(* IEC 61131-3 sources: LAxisCtrl/src/blocks (part 3) *)

                            ELSIF (_instCamIn.Error = TRUE) THEN
                                // Errorhandling
                                _status := AxisStatus#ERR_MC_CAMIN;
                                _statusText := STRING#'ERR_MC_CAMIN';
                                _errorAutoCleared := TRUE;
                                _diagnostics.subfunctionStatus := _instCamIn.ErrorId;
                                _subfunctionStatus := _instCamIn.ErrorId;
                                _diagnostics.basicMotionState := _basicMotionState;
                                _state := AXIS_STOP_ON_ERROR_SELECTION;
                                _basicMotionState := NO_SELECTION;
                            // ELSE
                            //   ; // Command selected
                            END_IF;

                            // Write MC_Command outputs to internal variable
                            _exeOfBasicMotion := 16#0;
                            _exeOfBasicMotion.%X0 := _instCamIn.Busy;
                            IF (_applicationMode = APPLICATION_MODE_ONCE) THEN
                                _exeOfBasicMotion.%X1 := _instCamIn.EndOfProfile;
                            END_IF;
                            _exeOfBasicMotion.%X2 := _instCamIn.CommandAborted;
                            _exeOfBasicMotion.%X3 := _instCamIn.Error;
                            _exeOfBasicMotion.%X6 := _instCamIn.StartSync;
                            _exeOfBasicMotion.%X7 := _instCamIn.InSync;
                            _exeOfBasicMotion.%X8 := _instCamIn.EndOfProfile;

                        GEAR_OUT_CAM_OUT_SELECTED:

                        // Firstcycle of command
                        IF (_firstCycleBasicMotion = TRUE) THEN
                            _applicativeBasicMotionError := FALSE;
                            _firstCycleBasicMotion := FALSE;

                            // Reset CAM_OUT command
                            _instCamOut(Slave := _refSyncAxis^,
                                        Execute := FALSE,
                                        SlavePosition := config.gearOutCamOut.slavePosition,
                                        SyncProfileReference := config.gearOutCamOut.syncProfileReference,
                                        MasterStopDistance := config.gearOutCamOut.masterStopDistance,
                                        Deceleration := config.gearOutCamOut.deceleration,
                                        Jerk := config.gearOutCamOut.jerk,
                                        SyncOutDirection := config.gearOutCamOut.syncOutDirection);

                            // Reset GEAR_OUT command
                            _instGearOut(Slave := _refSyncAxis^,
                                         Execute := FALSE,
                                         SlavePosition := config.gearOutCamOut.slavePosition,
                                         SyncProfileReference := config.gearOutCamOut.syncProfileReference,
                                         MasterStopDistance := config.gearOutCamOut.masterStopDistance,
                                         Deceleration := config.gearOutCamOut.deceleration,
                                         Jerk := config.gearOutCamOut.jerk,
                                         SyncOutDirection := config.gearOutCamOut.syncOutDirection);

                            CASE config.gearOutCamOut.gearOutCamOutMode OF
                                SYNCOUT_MODE_AUTOMATIC,
                                SYNCOUT_MODE_GEAROUT,
                                SYNCOUT_MODE_CAMOUT:
                                    // Get axis waiting function state
                                    IF (_typeAxis = SYNC_AXIS) THEN
                                        IF (_waitingFunctionStateAbortAutomatic < 0) // < 0: Automatic abort of waiting sync commands disabled
                                        THEN
                                            // Read waiting function state of axis
                                            _waitingFunctionState := _refSyncAxis^.StatusSynchronizedMotion.WaitingFunctionState;
                                        ELSE
                                            // Waiting function state already read out
                                            _waitingFunctionState := _waitingFunctionStateAbortAutomatic;
                                        END_IF;
                                        // Read function state of axis
                                        _functionState := _refSyncAxis^.StatusSynchronizedMotion.FunctionState;
                                    END_IF;

                                    _gearAndCamOutMode := config.gearOutCamOut.gearOutCamOutMode;
                                    _syncOutState := SYNCOUT_STATE_CHECK_WAITING; // Set next state

                                ELSE
                                    // Errorhandling - Invalid mode
                                    _status := AxisStatus#ERR_INVALID_GEAROUT_CAMOUT_MODE;
                                    _statusText := STRING#'ERR_INVALID_GEAROUT_CAMOUT_MODE';
                                    _errorAutoCleared := TRUE;
                                    _diagnostics.subfunctionStatus := WORD#0000;
                                    _subfunctionStatus := AxisStatus#STATUS_NO_CALL;
                                    _applicativeBasicMotionError := TRUE;
                                    // Set next state
                                    _state := AXIS_STOP_ON_ERROR_SELECTION;
                                    _basicMotionState := NO_SELECTION;
                            END_CASE;
                        END_IF;

                        IF (_applicativeBasicMotionError = FALSE) THEN
                            CASE _syncOutState OF
                                // ===========================================================
                                SYNCOUT_STATE_CHECK_WAITING:

                                    CASE _gearAndCamOutMode OF
                                        SYNCOUT_MODE_GEAROUT:
                                            CASE _waitingFunctionStateAbortAutomatic OF
                                                WFS_FS_CAMIN:
                                                    // Abort waiting camming in advance
                                                    _instCamOut.SyncProfileReference := CANCEL_ONLY_WAITING_GEARING_CAMMING;
                                                    _syncOutState := SYNCOUT_STATE_CAMOUT_WAITING_BUSY; // Set next state

                                                WFS_FS_GEARINPOS:
                                                    CASE config.gearOutCamOut.syncProfileReference OF
                                                        CANCEL_ONLY_WAITING_GEARING_CAMMING:
                                                            // Only gearOut - Set next state
                                                            _syncOutState := SYNCOUT_STATE_CHECK_ACTIVE;
                                                    ELSE
                                                        CASE _functionState OF
                                                            WFS_FS_GEARIN,
                                                            WFS_FS_GEARINPOS:
                                                                // Active gearing function
                                                                _syncOutState := SYNCOUT_STATE_CHECK_ACTIVE; // Set next state
                                                        ELSE
                                                            // Abort waiting gearing in advance
                                                            _instGearOut.SyncProfileReference := CANCEL_ONLY_WAITING_GEARING_CAMMING;
                                                            _syncOutState := SYNCOUT_STATE_GEAROUT_WAITING_BUSY; // Set next state
                                                        END_CASE;
                                                    END_CASE;

                                            ELSE
                                                // Only gearOut - Set next state
                                                _syncOutState := SYNCOUT_STATE_CHECK_ACTIVE;
                                            END_CASE;

                                        SYNCOUT_MODE_CAMOUT:
                                            CASE _waitingFunctionStateAbortAutomatic OF
                                                WFS_FS_GEARINPOS: // Waiting
                                                    // Abort waiting gearing in advance
                                                    _instGearOut.SyncProfileReference := CANCEL_ONLY_WAITING_GEARING_CAMMING;
                                                    _syncOutState := SYNCOUT_STATE_GEAROUT_WAITING_BUSY; // Set next state

                                                WFS_FS_CAMIN: // Waiting
                                                    CASE config.gearOutCamOut.syncProfileReference OF
                                                        CANCEL_ONLY_WAITING_GEARING_CAMMING:
                                                            // Only gearOut - Set next state
                                                            _syncOutState := SYNCOUT_STATE_CHECK_ACTIVE;
                                                    ELSE
                                                        CASE _functionState OF
                                                            WFS_FS_CAMIN: // Active
                                                                _syncOutState := SYNCOUT_STATE_CHECK_ACTIVE; // Set next state
                                                        ELSE
                                                            // Abort waiting camming in advance
                                                            _instCamOut.SyncProfileReference := CANCEL_ONLY_WAITING_GEARING_CAMMING;
                                                            _syncOutState := SYNCOUT_STATE_CAMOUT_WAITING_BUSY; // Set next state
                                                        END_CASE;
                                                    END_CASE;
                                            ELSE
                                                // Only camOut - Set next state
                                                _syncOutState := SYNCOUT_STATE_CHECK_ACTIVE;
                                            END_CASE;

                                        SYNCOUT_MODE_AUTOMATIC:
                                            CASE _waitingFunctionState OF
                                                WFS_FS_GEARINPOS, // Waiting
                                                WFS_FS_GEAROUT: // Waiting
                                                    CASE _functionState OF
                                                        WFS_FS_GEARIN, // Active
                                                        WFS_FS_GEARINPOS: // Active
                                                            ; // Gearing active - Waiting gearInPos will be aborted with MC_GEAROUT

                                                        WFS_FS_GEAROUT:
                                                            IF (_waitingFunctionStateAbortAutomatic < 0) THEN
                                                                ; // Automatic abort of waiting sync commands disabled
                                                            ELSE
                                                                // Automatic abort of waiting sync commands enabled - Separate call of MC_GearOut instruction is required
                                                                _instGearOut.SyncProfileReference := CANCEL_ONLY_WAITING_GEARING_CAMMING;
                                                            END_IF;
                                                    ELSE
                                                        _instGearOut.SyncProfileReference := CANCEL_ONLY_WAITING_GEARING_CAMMING;
                                                    END_CASE;
                                                    _functionState := -1;// Function state has to be updated at next use
                                                    _syncOutState := SYNCOUT_STATE_GEAROUT_WAITING_BUSY; // Set next state

                                                WFS_FS_CAMIN,  // Waiting
                                                WFS_FS_CAMOUT:  // Waiting
                                                    CASE _functionState OF
                                                        WFS_FS_CAMIN: // Active
                                                            ; // CamIn Active - Waiting CamIn will be aborted with MC_CAMOUT

                                                        WFS_FS_CAMOUT: // Active
                                                            IF (_waitingFunctionStateAbortAutomatic < 0) THEN
                                                                ; // Automatic abort of waiting sync commands disabled
                                                            ELSE
                                                                // Automatic abort of waiting sync commands enabled - Separate call of MC_CamOut instruction is required
                                                                _instCamOut.SyncProfileReference := CANCEL_ONLY_WAITING_GEARING_CAMMING;
                                                            END_IF;
                                                    ELSE
                                                        _instCamOut.SyncProfileReference := CANCEL_ONLY_WAITING_GEARING_CAMMING;
                                                    END_CASE;
                                                    _functionState := -1;// Function state has to be updated at next use
                                                    _syncOutState := SYNCOUT_STATE_CAMOUT_WAITING_BUSY; // Set next state

                                        ELSE
                                            // No waiting synchronous operation
                                            _syncOutState := SYNCOUT_STATE_CHECK_ACTIVE; // Set next state
                                        END_CASE;
                                    END_CASE;
                                    tempStateChangeActive := TRUE;

                                // ===========================================================
                                SYNCOUT_STATE_CHECK_ACTIVE:

                                    _instGearOut.SyncProfileReference := config.gearOutCamOut.syncProfileReference;
                                    _instCamOut.SyncProfileReference := config.gearOutCamOut.syncProfileReference;

                                    CASE _gearAndCamOutMode OF
                                        SYNCOUT_MODE_GEAROUT:
                                            _syncOutState := SYNCOUT_STATE_GEAROUT_ACTIVE_BUSY; // Set next state

                                        SYNCOUT_MODE_CAMOUT:
                                            _syncOutState := SYNCOUT_STATE_CAMOUT_ACTIVE_BUSY; // Set next state

                                        SYNCOUT_MODE_AUTOMATIC:
                                            CASE config.gearOutCamOut.syncProfileReference OF
                                                CANCEL_ONLY_WAITING_GEARING_CAMMING:
                                                    // No active synchronous operation
                                                    _syncOutState := SYNCOUT_STATE_DONE; // Set next state
                                            ELSE
                                                // Update function state of axis
                                                IF (_typeAxis = SYNC_AXIS) THEN
                                                    IF (_functionState < 0) THEN
                                                        _functionState := _refSyncAxis^.StatusSynchronizedMotion.FunctionState;
                                                    END_IF;
                                                END_IF;

                                                CASE _functionState OF
                                                    WFS_FS_GEAROUT,   // Active - Leads to error of MC_Instruction
                                                    WFS_FS_GEARIN,    // Active
                                                    WFS_FS_GEARINPOS: // Active
                                                        // Active gearing function
                                                        _syncOutState := SYNCOUT_STATE_GEAROUT_ACTIVE_BUSY; // Set next state

                                                    WFS_FS_CAMOUT, // Active - Leads to error of MC_Instruction
                                                    WFS_FS_CAMIN:  // Active
                                                        // Active camming function
                                                        _syncOutState := SYNCOUT_STATE_CAMOUT_ACTIVE_BUSY; // Set next state

                                                ELSE
                                                    // No active synchronous operation
                                                    _syncOutState := SYNCOUT_STATE_DONE; // Set next state
                                                END_CASE;
                                            END_CASE;

                                    END_CASE;
                                    tempStateChangeActive := TRUE;

                                // ===========================================================
                                SYNCOUT_STATE_GEAROUT_WAITING_BUSY,
                                SYNCOUT_STATE_GEAROUT_ACTIVE_BUSY:

                                    // Call MC_Instruction
                                    _instGearOut(Slave := _refSyncAxis^,
                                                Execute := TRUE);

                                    IF _instGearOut.Done THEN
                                        CASE _syncOutState OF
                                            SYNCOUT_STATE_GEAROUT_WAITING_BUSY:
                                            // Set next state
                                            _syncOutState := SYNCOUT_STATE_CHECK_ACTIVE;
                                            tempStateChangeActive := TRUE;

                                            SYNCOUT_STATE_GEAROUT_ACTIVE_BUSY:
                                            _syncOutState := SYNCOUT_STATE_DONE; // Set next state

                                        END_CASE;
                                        // Reset MC_Instruction
                                        _instGearOut(Slave := _refSyncAxis^,
                                                    Execute := FALSE);

                                    ELSIF _instGearOut.CommandAborted THEN
                                        _syncOutState := SYNCOUT_STATE_ABORTED; // Set next state
                                    END_IF;

                                // ===========================================================
                                SYNCOUT_STATE_CAMOUT_WAITING_BUSY,
                                SYNCOUT_STATE_CAMOUT_ACTIVE_BUSY:

                                    // Call MC_Instruction
                                    _instCamOut(Slave := _refSyncAxis^,
                                                Execute := TRUE);

                                    IF _instCamOut.Done THEN
                                        CASE _syncOutState OF
                                            SYNCOUT_STATE_CAMOUT_WAITING_BUSY:
                                                // Set next state
                                                _syncOutState := SYNCOUT_STATE_CHECK_ACTIVE;
                                                tempStateChangeActive := TRUE;

                                            SYNCOUT_STATE_CAMOUT_ACTIVE_BUSY:
                                                _syncOutState := SYNCOUT_STATE_DONE; // Set next state

                                        END_CASE;

                                        // Reset MC_Instruction
                                        _instCamOut(Slave := _refSyncAxis^,
                                                    Execute := FALSE);

                                    ELSIF _instCamOut.CommandAborted THEN
                                        _syncOutState := SYNCOUT_STATE_ABORTED; // Set next state
                                    END_IF;

                                // ===========================================================
                                SYNCOUT_STATE_DONE,
                                SYNCOUT_STATE_ABORTED,
                                SYNCOUT_STATE_ERROR:

                                    IF NOT _basicCommand.%X11 THEN
                                        // Return to NO_SELECTION if command finished
                                        _basicMotionState := NO_SELECTION;
                                    END_IF;

                            END_CASE;

                            IF _instGearOut.Error THEN
                                // Errorhandling
                                _status := AxisStatus#ERR_MC_GEAROUT;
                                _statusText := STRING#'ERR_MC_GEAROUT';
                                _errorAutoCleared := TRUE;
                                _diagnostics.subfunctionStatus := _instGearOut.ErrorId;
                                _subfunctionStatus := _instGearOut.ErrorId;
                                _diagnostics.basicMotionState := _basicMotionState;
                                _state := AXIS_STOP_ON_ERROR_SELECTION;
                                _basicMotionState := NO_SELECTION;

                                _syncOutState := SYNCOUT_STATE_ERROR; // Set next state

                            ELSIF _instCamOut.Error THEN
                                // Errorhandling
                                _status := AxisStatus#ERR_MC_CAMOUT;
                                _statusText := STRING#'ERR_MC_CAMOUT';
                                _errorAutoCleared := TRUE;
                                _diagnostics.subfunctionStatus := _instCamOut.ErrorId;
                                _subfunctionStatus := _instCamOut.ErrorId;
                                _diagnostics.basicMotionState := _basicMotionState;
                                _state := AXIS_STOP_ON_ERROR_SELECTION;
                                _basicMotionState := NO_SELECTION;

                                _syncOutState := SYNCOUT_STATE_ERROR; // Set next state
                            END_IF;

                            // Write MC_Command outputs to internal variable
                            _exeOfBasicMotion := 16#0;
                            _exeOfBasicMotion.%X0 := _syncOutState < SYNCOUT_STATE_DONE; // 7
                            _exeOfBasicMotion.%X1 := _syncOutState = SYNCOUT_STATE_DONE; // 7
                            _exeOfBasicMotion.%X2 := _syncOutState = SYNCOUT_STATE_ABORTED; // 8
                            _exeOfBasicMotion.%X3 := _syncOutState = SYNCOUT_STATE_ERROR; // 9
                            _exeOfBasicMotion.%X6 := _instCamOut.StartSyncOut OR _instGearOut.StartSyncOut;
                        END_IF;

                    ELSE
                        // Errorhandling
                        _status := AxisStatus#ERR_UNDEFINED_BASIC_MOTION_STATE;
                        _statusText := STRING#'ERR_UNDEFINED_BASIC_MOTION_STATE';
                        _errorUserCleared := TRUE;
                        _diagnostics.subfunctionStatus := WORD#0000;
                        _subfunctionStatus := AxisStatus#STATUS_NO_CALL;
                        // Set errorstate
                        _state := FB_ERROR;
                END_CASE;

                ABORT_WAITING_GEARINPOS_OR_CAMIN:
                    // Abort waiting absolute gearing / camIn job if new basic motion job is selected (config.generalSettings.abortWaitingSyncCmd = TRUE)

                    CASE _waitingFunctionStateAbortAutomatic OF
                        WFS_FS_GEARINPOS: // Waiting

                            _instGearOut(Slave := _refSyncAxis^,
                                         Execute := TRUE);

                            IF (_instGearOut.Done = TRUE) OR (_instGearOut.CommandAborted = TRUE)
                            THEN // Relative gearing command has aborted waiting absolute gearing job
                                _mainSelectionState := CALL_BASIC_MOTION; // Execute new basic motion command
                                tempStateChangeActive := TRUE;
                                _firstCycleBasicMotion := TRUE;

                            ELSIF (_instGearOut.Error = TRUE) THEN
                                _status := AxisStatus#ERR_MC_GEAROUT;
                                _statusText := STRING#'ERR_MC_GEAROUT';
                                _diagnostics.subfunctionStatus := _instGearOut.ErrorId;
                                _subfunctionStatus := _instGearOut.ErrorId;
                                // Errorhandling
                                _errorAutoCleared := TRUE;
                                // Set next state
                                _state := AXIS_STOP_ON_ERROR_SELECTION;
                                _mainSelectionState := CALL_BASIC_MOTION;
                                _basicMotionState := NO_SELECTION;
                            // ELSE
                            //   ; // Command running
                            END_IF;

                            // Write MC_Command outputs to internal variable
                            _exeOfBasicMotion := 16#0;
                            _exeOfBasicMotion.%X0 := _instGearOut.Busy;

                        WFS_FS_CAMIN: // Waiting

                            _instCamOut(Slave := _refSyncAxis^,
                                        Execute := TRUE);

                            IF (_instCamOut.Done = TRUE) OR (_instCamOut.CommandAborted = TRUE)
                            THEN
                                _mainSelectionState := CALL_BASIC_MOTION; // Execute new basic motion command
                                tempStateChangeActive := TRUE;
                                _firstCycleBasicMotion := TRUE;

                            ELSIF (_instCamOut.Error = TRUE) THEN
                                _status := AxisStatus#ERR_MC_CAMOUT;
                                _statusText := STRING#'ERR_MC_CAMOUT';
                                _diagnostics.subfunctionStatus := _instCamOut.ErrorId;
                                _subfunctionStatus := _instCamOut.ErrorId;
                                // Errorhandling
                                _errorAutoCleared := TRUE;
                                // Set next state
                                _state := AXIS_STOP_ON_ERROR_SELECTION;
                                _mainSelectionState := CALL_BASIC_MOTION;
                                _basicMotionState := NO_SELECTION;
                            // ELSE
                            //   ; // Command running
                            END_IF;

                            // Write MC_Command outputs to internal variable
                            _exeOfBasicMotion := 16#0;
                            _exeOfBasicMotion.%X0 := _instCamOut.Busy;

                    END_CASE;
                ELSE
                    // Errorhandling
                    _status := AxisStatus#ERR_UNDEFINED_MAIN_SELECTION_STATE;
                    _statusText := STRING#'ERR_UNDEFINED_MAIN_SELECTION_STATE';
                    _errorUserCleared := TRUE;
                    _diagnostics.subfunctionStatus := WORD#0000;
                    _subfunctionStatus := AxisStatus#STATUS_NO_CALL;
                    // Set errorstate
                    _state := FB_ERROR;
            END_CASE;

        UNTIL (tempStateChangeActive = FALSE)
        END_REPEAT;

        //----------------------------------------------------------------------------------------------
        // Execution of homing functionality
        //----------------------------------------------------------------------------------------------

        // Statemachine for homing functionality
        CASE _passiveHomingState OF
            // Selection of extended homing mode
            NO_HOMING_ACTIVE:
                ; // Do nothing

            STANDARD_HOMING:
                // No additional features

                // Firstcycle of command
                IF (_firstCycleHoming = TRUE) THEN
                    // Reset MC_HOME command
                    _instHome(Axis := _refAxis^,
                            Execute := FALSE,
                            Position := config.homing.position,
                            Mode := config.homing.mode,
                            Sensor := config.homing.sensor);

                    IF (_basicMotionState = ACTIVE_HOMING_SELECTED) THEN
                        _basicMotionState := NO_SELECTION;
                    END_IF;
                END_IF;

                // Call MC_Command
                _instHome(Axis := _refAxis^,
                          Execute := _extendedCommand.%X2); // Input: homing

                // Evaluate MC_Command
                IF (_instHome.Busy = FALSE) AND
                    (_instHome.Done = FALSE) AND
                    (_instHome.CommandAborted = FALSE) AND
                    (_instHome.Error = FALSE)
                THEN
                    // Return to NO_SELECTION if command finished
                    _passiveHomingState := NO_HOMING_ACTIVE;

                ELSIF (_instHome.Error = TRUE) THEN
                    // Errorhandling
                    _status := AxisStatus#ERR_MC_HOME;
                    _statusText := STRING#'ERR_MC_HOME';
                    _errorAutoCleared := TRUE;
                    _diagnostics.subfunctionStatus := _instHome.ErrorId;
                    _subfunctionStatus := _instHome.ErrorId;
                    _passiveHomingState := NO_HOMING_ACTIVE;
                    // Set next state
                    _state := AXIS_STOP_ON_ERROR_SELECTION;
                    // ELSE
                    //   ; // Command selected
                END_IF;
                _exeOfHoming := 16#0;
                _exeOfHoming.%X0 := _instHome.Busy;
                _exeOfHoming.%X1 := _instHome.Done;
                _exeOfHoming.%X2 := _instHome.CommandAborted;
                _exeOfHoming.%X3 := _instHome.Error;

            ELSE
                // Errorhandling
                _status := AxisStatus#ERR_INVALID_HOMING_EXTENDED_MODE;
                _statusText := STRING#'ERR_INVALID_HOMING_EXTENDED_MODE';
                _errorAutoCleared := TRUE;
                _diagnostics.subfunctionStatus := WORD#0000;
                _subfunctionStatus := AxisStatus#STATUS_NO_CALL;
                _diagnostics.basicMotionState := _basicMotionState;
                _diagnostics.superimposedMotionState := _supImpMotionState;
                // Set next state
                _state := AXIS_STOP_ON_ERROR_SELECTION;
                _basicMotionState := NO_SELECTION;
                _passiveHomingState := NO_HOMING_ACTIVE;
        END_CASE;

        //----------------------------------------------------------------------------------------------
        // Execution of functionalities of superimposed coordinate system
        //----------------------------------------------------------------------------------------------

        // Statemachine for superimposed motion commands
        // Write diagnostics
        _diagnostics.basicMotionState := _basicMotionState;
        _diagnostics.superimposedMotionState := _supImpMotionState;

        CASE _supImpMotionState OF
            NO_SELECTION:
                ; // Do nothing

            POS_SUPERIMPOSED_SELECTED:
                // Additional features (applicative) : Specified direction

                // Firstcycle of command
                IF (_firstCycleSupImpMotion = TRUE) THEN
                    // Configurate the direction of rotation
                    IF ((config.posSuperimposed.direction = 0) AND (config.posSuperimposed.distance >= 0.0))  // Sign of distance is evaluated
                        OR (config.posSuperimposed.direction = FORWARD_DIR)// Positive direction
                    THEN
                        _supImpMotionPosition := Abs(config.posSuperimposed.distance);
                        // Reset MC_MOVESUPERIMPOSED command
                        _instMoveSuperimposed(Axis := _refPosAxis^,
                                              Execute := FALSE,
                                              Distance := _supImpMotionPosition,
                                              VelocityDiff := config.posSuperimposed.velocityDiff,
                                              Acceleration := config.posSuperimposed.acceleration,
                                              Deceleration := config.posSuperimposed.deceleration,
                                              Jerk := config.posSuperimposed.jerk);

                        _applicativeSupImpMotionError := FALSE;

                    ELSIF ((config.posSuperimposed.direction = 0) AND (config.posSuperimposed.distance < 0.0)) // Sign of distance is evaluated
                        OR (config.posSuperimposed.direction = BACKWARD_DIR)// Negative direction
                    THEN
                        _supImpMotionPosition := -Abs(config.posSuperimposed.distance);
                        // Reset MC_MOVESUPERIMPOSED command
                        _instMoveSuperimposed(Axis := _refPosAxis^,
                                                Execute := FALSE,
                                                Distance := _supImpMotionPosition,
                                                VelocityDiff := config.posSuperimposed.velocityDiff,
                                                Acceleration := config.posSuperimposed.acceleration,
                                                Deceleration := config.posSuperimposed.deceleration,
                                                Jerk := config.posSuperimposed.jerk);

                        _applicativeSupImpMotionError := FALSE;

                    ELSE
                        // Errorhandling - Invalid direction
                        _status := AxisStatus#ERR_INVALID_POS_SUPERIMPOSED_DIR;
                        _statusText := STRING#'ERR_INVALID_POS_SUPERIMPOSED_DIR';
                        _errorAutoCleared := TRUE;
                        _diagnostics.subfunctionStatus := WORD#0000;
                        _subfunctionStatus := AxisStatus#STATUS_NO_CALL;
                        _applicativeSupImpMotionError := TRUE;
                        // Set next state
                        _state := AXIS_STOP_ON_ERROR_SELECTION;
                        _supImpMotionState := NO_SELECTION;
                    END_IF;
                END_IF;

                IF (_applicativeSupImpMotionError = FALSE) THEN
                    // Call MC_Command
                    _instMoveSuperimposed(Axis := _refPosAxis^,
                                          Execute := _supImpCommand.%X0); // Input: posSuperimposed

                    // Evaluate MC_Command
                    IF (_instMoveSuperimposed.Busy = FALSE) AND
                        (_instMoveSuperimposed.Error = FALSE) AND
                        (_instMoveSuperimposed.Done = FALSE) AND
                        (_instMoveSuperimposed.CommandAborted = FALSE)
                    THEN
                        // Return to NO_SELECTION if command finished
                        _supImpMotionState := NO_SELECTION;

                    ELSIF (_instMoveSuperimposed.Error = TRUE) THEN
                        // Errorhandling
                        _status := AxisStatus#ERR_MC_MOVESUPERIMPOSED;
                        _statusText := STRING#'ERR_MC_MOVESUPERIMPOSED';
                        _errorAutoCleared := TRUE;
                        _diagnostics.subfunctionStatus := _instMoveSuperimposed.ErrorId;
                        _subfunctionStatus := _instMoveSuperimposed.ErrorId;
                        // Set next state
                        _state := AXIS_STOP_ON_ERROR_SELECTION;
                        _supImpMotionState := NO_SELECTION;
                    // ELSE
                    //   ; // command selected
                    END_IF;
                    _exeOfSupImpMotionState := 16#0;
                    _exeOfSupImpMotionState.%X0 := _instMoveSuperimposed.Busy;
                    _exeOfSupImpMotionState.%X1 := _instMoveSuperimposed.Done;
                    _exeOfSupImpMotionState.%X2 := _instMoveSuperimposed.CommandAborted;
                    _exeOfSupImpMotionState.%X3 := _instMoveSuperimposed.Error;
                    _exeOfSupImpMotionState.%X4 := _instMoveSuperimposed.Busy;
                END_IF;

            HALT_SUPERIMPOSED_SELECTED:

                // Firstcycle of command
                IF (_firstCycleSupImpMotion = TRUE) THEN
                    _instHaltSuperimposed(Axis := _refPosAxis^,
                                          Execute := FALSE,
                                          Deceleration := config.haltSuperimposed.deceleration,
                                          Jerk := config.haltSuperimposed.jerk,
                                          AbortAcceleration := config.haltSuperimposed.abortAcceleration);
                END_IF;

                // Call MC_Command
                _instHaltSuperimposed(Axis := _refPosAxis^,
                                      Execute := _supImpCommand.%X3); // Input: haltSuperimposed

                // Evaluate MC_Command
                IF (_instHaltSuperimposed.Busy = FALSE) AND
                    (_instHaltSuperimposed.Error = FALSE) AND
                    (_instHaltSuperimposed.Done = FALSE) AND
                    (_instHaltSuperimposed.CommandAborted = FALSE)
                THEN
                    // Return to NO_SELECTION if command finished
                    _supImpMotionState := NO_SELECTION;

                ELSIF (_instHaltSuperimposed.Error = TRUE) THEN
                    // Errorhandling
                    _status := AxisStatus#ERR_MC_HALTSUPERIMPOSED;
                    _statusText := STRING#'ERR_MC_HALTSUPERIMPOSED';
                    _errorAutoCleared := TRUE;
                    _diagnostics.subfunctionStatus := _instHaltSuperimposed.ErrorId;
                    _subfunctionStatus := _instHaltSuperimposed.ErrorId;
                    // Set next state
                    _state := AXIS_STOP_ON_ERROR_SELECTION;
                    _supImpMotionState := NO_SELECTION;
                    // ELSE
                    //   ; // command selected
                END_IF;
                _exeOfSupImpMotionState := 16#0;
                _exeOfSupImpMotionState.%X0 := _instHaltSuperimposed.Busy;
                _exeOfSupImpMotionState.%X1 := _instHaltSuperimposed.Done;
                _exeOfSupImpMotionState.%X2 := _instHaltSuperimposed.CommandAborted;
                _exeOfSupImpMotionState.%X3 := _instHaltSuperimposed.Error;
                _exeOfSupImpMotionState.%X4 := _instHaltSuperimposed.Busy;

            PHASING_SELECTED:
                // Additional features (applicative) : Change setpoint on the fly (phaseShift)

                // Firstcycle of command
                IF (_firstCycleSupImpMotion = TRUE) THEN
                    // Reset MC_PHASING_ABSOLUTE command
                    _instPhasingAbsolute(Master := _refMasterAxis^,
                                         Slave := _refSyncAxis^,
                                         Execute := FALSE);

                    // Reset MC_PHASING_RELATIVE command
                    _instPhasingRelative(Master := _refMasterAxis^,
                                         Slave := _refSyncAxis^,
                                         Execute := FALSE);

                    _instPhasingAbsolute.PhaseShift := config.phasing.phaseShift;
                    _instPhasingRelative.PhaseShift := config.phasing.phaseShift;
                    _phaseShift := config.phasing.phaseShift;

                    _instPhasingAbsolute.Velocity := config.phasing.velocity;
                    _instPhasingRelative.Velocity := config.phasing.velocity;
                    _instPhasingAbsolute.Acceleration := config.phasing.acceleration;
                    _instPhasingRelative.Acceleration := config.phasing.acceleration;
                    _instPhasingAbsolute.Deceleration := config.phasing.deceleration;
                    _instPhasingRelative.Deceleration := config.phasing.deceleration;
                    _instPhasingAbsolute.Jerk := config.phasing.jerk;
                    _instPhasingRelative.Jerk := config.phasing.jerk;
                    _instPhasingAbsolute.ProfileReference := config.phasing.profileReference;
                    _instPhasingRelative.ProfileReference := config.phasing.profileReference;
                    _instPhasingAbsolute.PhasingDistance := config.phasing.phasingDistance;
                    _instPhasingRelative.PhasingDistance := config.phasing.phasingDistance;
                    _instPhasingAbsolute.StartPosition := config.phasing.startPosition;
                    _instPhasingRelative.StartPosition := config.phasing.startPosition;
                    _instPhasingAbsolute.Direction := config.phasing.direction;
                    _instPhasingRelative.Direction := config.phasing.direction;

                    _phaseAbsolute := config.phasing.phaseAbsolute;
                    _changePhaseShiftOnTheFly := config.phasing.phaseShiftChangeOnTheFly;

                ELSIF ((_changePhaseShiftOnTheFly = TRUE) AND
                    (config.phasing.phaseShift <> _phaseShift))
                    AND (_phaseAbsolute = TRUE)
                    AND (_instPhasingAbsolute.CommandAborted = FALSE)
                THEN
                    // Reset MC_PHASING_ABSOLUTE command - Phaseshift on the fly is only possible at phasing absolute
                    _instPhasingAbsolute(Master := _refMasterAxis^,
                                         Slave := _refSyncAxis^,
                                         Execute := FALSE);

                    _instPhasingAbsolute.PhaseShift := config.phasing.phaseShift;
                    _phaseShift := config.phasing.phaseShift;

                    // Copy also Dynamics
                    _instPhasingAbsolute.Velocity := config.phasing.velocity;
                    _instPhasingAbsolute.Acceleration := config.phasing.acceleration;
                    _instPhasingAbsolute.Deceleration := config.phasing.deceleration;
                    _instPhasingAbsolute.Jerk := config.phasing.jerk;
                    _instPhasingAbsolute.ProfileReference := config.phasing.profileReference;
                    _instPhasingAbsolute.PhasingDistance := config.phasing.phasingDistance;
                    _instPhasingAbsolute.StartPosition := config.phasing.startPosition;
                    _instPhasingAbsolute.Direction := config.phasing.direction;
                END_IF;

                // Select phasing absolute or relative
                IF (_phaseAbsolute = TRUE) THEN
                    // Absolute phasing
                    // Call MC_Command
                    _instPhasingAbsolute(Master := _refMasterAxis^,
                                         Slave := _refSyncAxis^,
                                         Execute := _supImpCommand.%X1); // Input: phasing
                    // Evaluate MC_Command
                    IF (_instPhasingAbsolute.Busy = FALSE) AND
                        (_instPhasingAbsolute.Error = FALSE) AND
                        (_instPhasingAbsolute.Done = FALSE) AND
                        (_instPhasingAbsolute.CommandAborted = FALSE)
                    THEN
                        // Return to NO_SELECTION if command finished
                        _supImpMotionState := NO_SELECTION;

                    ELSIF (_instPhasingAbsolute.Error = TRUE) THEN
                        // Errorhandling
                        _status := AxisStatus#ERR_MC_PHASINGABSOLUTE;
                        _statusText := STRING#'ERR_MC_PHASINGABSOLUTE';
                        _errorAutoCleared := TRUE;
                        _diagnostics.subfunctionStatus := WORD#0000;
                        _subfunctionStatus := _instPhasingAbsolute.ErrorId;
                        _changePhaseShiftOnTheFly := FALSE;
                        // Set next state
                        _state := AXIS_STOP_ON_ERROR_SELECTION;
                        _supImpMotionState := NO_SELECTION;
                    // ELSE
                    //   ; // Command busy
                    END_IF;
                    _exeOfSupImpMotionState := 16#0;
                    _exeOfSupImpMotionState.%X0 := _instPhasingAbsolute.Busy;
                    _exeOfSupImpMotionState.%X1 := _instPhasingAbsolute.Done;
                    _exeOfSupImpMotionState.%X2 := _instPhasingAbsolute.CommandAborted;
                    _exeOfSupImpMotionState.%X3 := _instPhasingAbsolute.Error;
                    _exeOfSupImpMotionState.%X4 := _instPhasingAbsolute.StartPhasing;
                ELSE
                    // Relative phasing
                    // Call MC_Command
                    _instPhasingRelative(Master := _refMasterAxis^,
                                         Slave := _refSyncAxis^,
                                         Execute := _supImpCommand.%X1); // Input: phasing

                    // Evaluate MC_Command
                    IF (_instPhasingRelative.Busy = FALSE) AND
                        (_instPhasingRelative.Error = FALSE) AND
                        (_instPhasingRelative.Done = FALSE) AND
                        (_instPhasingRelative.CommandAborted = FALSE)
                    THEN
                        // Return to NO_SELECTION if command finished
                        _supImpMotionState := NO_SELECTION;

                    ELSIF (_instPhasingRelative.Error = TRUE) THEN
                        // Errorhandling
                        _status := AxisStatus#ERR_MC_PHASINGRELATIVE;
                        _statusText := STRING#'ERR_MC_PHASINGRELATIVE';
                        _errorAutoCleared := TRUE;
                        _diagnostics.subfunctionStatus := _instPhasingRelative.ErrorId;
                        _subfunctionStatus := _instPhasingRelative.ErrorId;
                        _changePhaseShiftOnTheFly := FALSE;
                        // Set next state
                        _state := AXIS_STOP_ON_ERROR_SELECTION;
                        _supImpMotionState := NO_SELECTION;
                    // ELSE
                    //   ; // Command selected
                    END_IF;
                    _exeOfSupImpMotionState := 16#0;
                    _exeOfSupImpMotionState.%X0 := _instPhasingRelative.Busy;
                    _exeOfSupImpMotionState.%X1 := _instPhasingRelative.Done;
                    _exeOfSupImpMotionState.%X2 := _instPhasingRelative.CommandAborted;
                    _exeOfSupImpMotionState.%X3 := _instPhasingRelative.Error;
                    _exeOfSupImpMotionState.%X4 := _instPhasingRelative.StartPhasing;
                END_IF;

            OFFSET_SELECTED:

                // Firstcycle of command
                IF (_firstCycleSupImpMotion = TRUE) THEN
                    // Reset MC_OFFSET_ABSOLUTE command
                    _instOffsetAbsolute(Slave := _refSyncAxis^,
                                        Execute := FALSE);

                    // Reset MC_OFFSET_RELATIVE command
                    _instOffsetRelative(Slave := _refSyncAxis^,
                                        Execute := FALSE);

                    _instOffsetAbsolute.Offset := config.offset.offset;
                    _instOffsetRelative.Offset := config.offset.offset;
                    _offsetValue := config.offset.offset;

                    _instOffsetAbsolute.ProfileReference := config.offset.profileReference;
                    _instOffsetRelative.ProfileReference := config.offset.profileReference;
                    _instOffsetAbsolute.OffsetDistance := config.offset.offsetDistance;
                    _instOffsetRelative.OffsetDistance := config.offset.offsetDistance;
                    _instOffsetAbsolute.StartPosition := config.offset.startPosition;
                    _instOffsetRelative.StartPosition := config.offset.startPosition;
                    _instOffsetAbsolute.Direction := config.offset.direction;
                    _instOffsetRelative.Direction := config.offset.direction;

                    _offsetAbsolute := config.offset.offsetAbsolute;
                    _changeOffsetOnTheFly := config.offset.offsetChangeOnTheFly;

                ELSIF ((_changeOffsetOnTheFly = TRUE) AND
                    (config.offset.offset <> _offsetValue))
                    AND (_offsetAbsolute = TRUE)
                    AND (_instOffsetAbsolute.CommandAborted = FALSE)
                THEN
                    // Reset MC_OFFSET_ABSOLUTE command - Offset on the fly is only possible at offset absolute
                    _instOffsetAbsolute(Slave := _refSyncAxis^,
                                        Execute := FALSE);

                    _instOffsetAbsolute.Offset := config.offset.offset;
                    _offsetValue := config.offset.offset;
                END_IF;

                // Select offset absolute or relative
                IF (_offsetAbsolute = TRUE) THEN
                    // Absolute phasing
                    // Call MC_Command
                    _instOffsetAbsolute(Slave := _refSyncAxis^,
                                        Execute := _supImpCommand.%X2); // Input: offset

                    // Evaluate MC_Command
                    IF (_instOffsetAbsolute.Busy = FALSE) AND
                        (_instOffsetAbsolute.Error = FALSE) AND
                        (_instOffsetAbsolute.Done = FALSE) AND
                        (_instOffsetAbsolute.CommandAborted = FALSE)
                    THEN
                        // Return to NO_SELECTION if command finished
                        _supImpMotionState := NO_SELECTION;

                    ELSIF (_instOffsetAbsolute.Error = TRUE) THEN
                        // Errorhandling
                        _status := AxisStatus#ERR_MC_OFFSETABSOLUTE;
                        _statusText := STRING#'ERR_MC_OFFSETABSOLUTE';
                        _errorAutoCleared := TRUE;
                        _diagnostics.subfunctionStatus := _instOffsetAbsolute.ErrorId;
                        _subfunctionStatus := _instOffsetAbsolute.ErrorId;
                        _changeOffsetOnTheFly := FALSE;
                        // Set next state
                        _state := AXIS_STOP_ON_ERROR_SELECTION;
                        _supImpMotionState := NO_SELECTION;
                    // ELSE
                    //   ; // Command busy
                    END_IF;
                    _exeOfSupImpMotionState := 16#0;
                    _exeOfSupImpMotionState.%X0 := _instOffsetAbsolute.Busy;
                    _exeOfSupImpMotionState.%X1 := _instOffsetAbsolute.Done;
                    _exeOfSupImpMotionState.%X2 := _instOffsetAbsolute.CommandAborted;
                    _exeOfSupImpMotionState.%X3 := _instOffsetAbsolute.Error;
                    _exeOfSupImpMotionState.%X4 := _instOffsetAbsolute.StartOffset;
                ELSE
                    // Relative offset
                    // Call MC_Command
                    _instOffsetRelative(Slave := _refSyncAxis^,
                                        Execute := _supImpCommand.%X2); // Input: offset

                    // Evaluate MC_Command
                    IF (_instOffsetRelative.Busy = FALSE) AND
                        (_instOffsetRelative.Error = FALSE) AND
                        (_instOffsetRelative.Done = FALSE) AND
                        (_instOffsetRelative.CommandAborted = FALSE)
                    THEN
                        // Return to NO_SELECTION if command finished
                        _supImpMotionState := NO_SELECTION;

                    ELSIF (_instOffsetRelative.Error = TRUE) THEN
                        // Errorhandling
                        _status := AxisStatus#ERR_MC_OFFSETRELATIVE;
                        _statusText := STRING#'ERR_MC_OFFSETRELATIVE';
                        _errorAutoCleared := TRUE;
                        _diagnostics.subfunctionStatus := _instOffsetRelative.ErrorId;
                        _subfunctionStatus := _instOffsetRelative.ErrorId;
                        _changeOffsetOnTheFly := FALSE;
                        // Set next state
                        _state := AXIS_STOP_ON_ERROR_SELECTION;
                        _supImpMotionState := NO_SELECTION;
                    // ELSE
                    //   ; // Command selected
                    END_IF;
                    _exeOfSupImpMotionState := 16#0;
                    _exeOfSupImpMotionState.%X0 := _instOffsetRelative.Busy;
                    _exeOfSupImpMotionState.%X1 := _instOffsetRelative.Done;
                    _exeOfSupImpMotionState.%X2 := _instOffsetRelative.CommandAborted;
                    _exeOfSupImpMotionState.%X3 := _instOffsetRelative.Error;
                    _exeOfSupImpMotionState.%X4 := _instOffsetRelative.StartOffset;
                END_IF;

            ELSE
                // Errorhandling
                _status := AxisStatus#ERR_UNDEFINED_SUPERIMPOSED_MOTION_STATE;
                _statusText := STRING#'ERR_UNDEFINED_SUPERIMPOSED_MOTION_STATE';
                _errorUserCleared := TRUE;
                _diagnostics.subfunctionStatus := WORD#0000;
                _subfunctionStatus := AxisStatus#STATUS_NO_CALL;
                // Set errorstate
                _state := FB_ERROR;
        END_CASE;

        //----------------------------------------------------------------------------------------------
        // Execution of torquelimiting functionality
        //----------------------------------------------------------------------------------------------

        // Statemachine for torquelimiting
        REPEAT
            tempStateChangeActive := FALSE;
            CASE _torqueLimitingState OF
                NO_TORQUE_LIMITING_ACTIVE:
                    ;

                TORQUE_LIMITING_DISABLE:
                    // Torquelimiting disable
                    _instTorqueLimiting(Axis := _refSpeedAxis^,
                                        Enable := FALSE);

                    // Check state of torque limiting
                    IF (_instTorqueLimiting.Busy = FALSE) THEN
                        // set next state
                        _torqueLimitingState := NO_TORQUE_LIMITING_ACTIVE;
                    // ELSE
                        //   ; // Waiting for MC_TorqueLimiting is not busy
                    END_IF;

                TORQUE_LIMITING_SELECTED:
                    // No extended homing function active
                    _instTorqueLimiting(Axis := _refSpeedAxis^,
                                        Enable := _extendedCommand.%X1,
                                        Limit := config.torqueLimiting.limit,
                                        Mode := config.torqueLimiting.mode);

                    IF (_instTorqueLimiting.Busy = FALSE) THEN
                        // Reset state
                        _torqueLimitingState := NO_TORQUE_LIMITING_ACTIVE;
                    END_IF;

                FIXED_STOP_DETECTION_ACTIVE:
                    // Extended homing function active
                    _instTorqueLimiting(Axis := _refSpeedAxis^,
                                        Enable := TRUE,
                                        Limit := config.homing.extendedModeTorqueLimit, // Always use configured value
                                        Mode := MODE_FIXED_STOP_DETECTION);

                    IF ((_homingSubState = HOMING_IDLE) AND (_basicMotionState = ACTIVE_HOMING_SELECTED)) THEN
                        // Fixed stop process has finished - Axis is still in clamping
                        _torqueLimitingState := FIXED_STOP_DETECTION_FINISHED;
                        tempStateChangeActive := TRUE;
                    ELSIF (_basicMotionState <> ACTIVE_HOMING_SELECTED) THEN
                        // Error occurred - change state depending on inClamping
                        IF (_instTorqueLimiting.InClamping = TRUE) THEN
                            // Axis is in clamping
                            _torqueLimitingState := FIXED_STOP_DETECTION_ERROR_IN_CLAMPING;
                            tempStateChangeActive := TRUE;
                        ELSE
                            // Axis is in not clamping
                            _torqueLimitingState := FIXED_STOP_DETECTION_ERROR_NOT_IN_CLAMPING;
                            tempStateChangeActive := TRUE;
                        END_IF;
                    // ELSE
                    //   ; // Fixed stop detection is running
                    END_IF;

                FIXED_STOP_DETECTION_FINISHED:
                    // Homing on fixed stop process has finished
                    _instTorqueLimiting(Axis := _refSpeedAxis^,
                                        Enable := TRUE,
                                        Limit := config.homing.extendedModeTorqueLimit, // Always use configured value
                                        Mode := MODE_FIXED_STOP_DETECTION);

                    IF (_instTorqueLimiting.InClamping = FALSE) THEN
                        // InClamping = FALSE
                        IF (_extendedCommand.%X1 = TRUE) // Torquelimiting
                        THEN
                            _torqueLimitingState := TORQUE_LIMITING_SELECTED;
                        ELSE
                            _torqueLimitingState := TORQUE_LIMITING_DISABLE;
                        END_IF;
                        tempStateChangeActive := TRUE;
                    ELSE
                        // InClamping = TRUE
                        IF (_extendedCommand.%X1 = TRUE) // Torquelimiting
                            AND (config.torqueLimiting.mode = MODE_FIXED_STOP_DETECTION)
                        THEN
                            // Change State
                            _torqueLimitingState := TORQUE_LIMITING_SELECTED;
                            tempStateChangeActive := TRUE;
                        // ELSE
                        //   ; // Wait for inClamping = FALSE
                        END_IF;
                    END_IF;

                FIXED_STOP_DETECTION_ERROR_IN_CLAMPING:
                    // Errorstate, torquelimiting is still active and axis not in clamping
                    _instTorqueLimiting(Axis := _refSpeedAxis^,
                                        Enable := TRUE,
                                        Limit := config.homing.extendedModeTorqueLimit, // Always use configured value
                                        Mode := MODE_FIXED_STOP_DETECTION);

                    IF (_instTorqueLimiting.InClamping = FALSE) THEN
                        // InClamping = FALSE -> reset torque limiting state
                        _torqueLimitingState := TORQUE_LIMITING_DISABLE;
                        // Torquelimiting disable
                        tempStateChangeActive := TRUE;
                    END_IF;

                FIXED_STOP_DETECTION_ERROR_NOT_IN_CLAMPING:
                    // Errorstate, torquelimiting is still active and axis in clamping
                    _instTorqueLimiting(Axis := _refSpeedAxis^,
                                        Enable := TRUE,
                                        Limit := config.homing.extendedModeTorqueLimit, // Always use configured value
                                        Mode := MODE_FIXED_STOP_DETECTION);

                    IF (_instTorqueLimiting.InClamping = TRUE) THEN
                        // InClamping = TRUE -> change state
                        _torqueLimitingState := FIXED_STOP_DETECTION_ERROR_IN_CLAMPING;
                        tempStateChangeActive := TRUE;

                    ELSIF (_basicMotionState <> NO_SELECTION)
                        OR (_supImpMotionState <> NO_SELECTION)
                        OR (_passiveHomingState <> NO_HOMING_ACTIVE)
                    THEN
                        // New valid command is set -> reset error state
                        _torqueLimitingState := TORQUE_LIMITING_DISABLE;
                        tempStateChangeActive := TRUE;
                    // ELSE
                    //   ; // Waiting for new command or axis is getting in clamping
                    END_IF;
                ELSE
                    // Errorhandling
                    _status := AxisStatus#ERR_UNDEFINED_TORQUE_LIMITING_STATE;
                    _statusText := STRING#'ERR_UNDEFINED_TORQUE_LIMITING_STATE';
                    _errorUserCleared := TRUE;
                    _diagnostics.basicMotionState := _basicMotionState;
                    _diagnostics.superimposedMotionState := _supImpMotionState;
                    _diagnostics.subfunctionStatus := WORD#0000;
                    _subfunctionStatus := AxisStatus#STATUS_NO_CALL;
                    // Set errorstate
                    _state := FB_ERROR;
            END_CASE;
        UNTIL (tempStateChangeActive = FALSE)
        END_REPEAT;

        // Evaluate MC_Command
        IF (_instTorqueLimiting.Error = TRUE) AND ((_torqueLimitingErrorOld = FALSE) OR (_status = AxisStatus#STATUS_SUBSEQUENT_CALL)) THEN
            // Errorhandling
            _status := AxisStatus#ERR_MC_TORQUELIMITING;
            _statusText := STRING#'ERR_MC_TORQUELIMITING';
            _errorAutoCleared := TRUE;
            _diagnostics.basicMotionState := _basicMotionState;
            _diagnostics.superimposedMotionState := _supImpMotionState;
            _diagnostics.subfunctionStatus := _instTorqueLimiting.ErrorId;
            _subfunctionStatus := _instTorqueLimiting.ErrorId;

            _state := AXIS_STOP_ON_ERROR_SELECTION;

        ELSIF (_instTorqueLimiting.Error = FALSE) AND ((_torqueLimitingErrorOld = TRUE) AND (_status = AxisStatus#ERR_MC_TORQUELIMITING)) THEN
            _status := AxisStatus#STATUS_SUBSEQUENT_CALL;
            _statusText := STRING#'STATUS_SUBSEQUENT_CALL';
            _errorAutoCleared := FALSE;
        END_IF;

        _torqueLimitingErrorOld := _instTorqueLimiting.Error;

        //----------------------------------------------------------------------------------------------
        // Selection of StopOnError / implementation of fastStop
        //----------------------------------------------------------------------------------------------

        // Check for stopping if error occurred during execution of motion commands
        IF (_state = AXIS_STOP_ON_ERROR_SELECTION) THEN
            _basicMotionState := NO_SELECTION;
            _supImpMotionState := NO_SELECTION;
            _passiveHomingState := NO_HOMING_ACTIVE;

            IF (config.generalSettings.stopOnError = TRUE) THEN
                // Evaluate error
                IF tempStatusWord.%X0 THEN
                    // Axis enabled
                    IF (tempStatusWord.%X1 = TRUE) THEN
                        // TO Alarm present
                        _state := AXIS_MOTION;
                    ELSE
                        _stopWithoutSignalization := TRUE;
                        _firstCycleBasicMotion := TRUE;
                        _state := AXIS_STOP_ON_ERROR_EXECUTION;
                    END_IF;
                ELSE
                // Axis disabled
                _state := AXIS_MOTION;
                END_IF;
            ELSE
                // Dont StopOnError
                _state := AXIS_MOTION;
            END_IF;
        END_IF;

        // Implementation of fastStop
        IF _stopWithoutSignalization
            OR
            (
            TRUE
            AND (_basicMotionState = FAST_STOP_SELECTED)
            AND (_mainSelectionState = CALL_BASIC_MOTION)
            )
        THEN
            // Additional feature: Load emergency stop dynamics (TO) if no valid dynamics are configured for fastStop

            // Firstcycle of command
            IF (_firstCycleBasicMotion = TRUE) THEN
                // Reset HALT command
                _instHalt(Axis := _refSpeedAxis^,
                          Execute := FALSE,
                          Mode := 0); // Mode := 0 "The basic motion and the superimposed motion are stopped." MC_Halt instance is also used for input 'stop', where the 'haltMode' can now be specified via config

                _firstCycleDone := TRUE;
                // Check dynamics for fastStop
                // Load TO emergency Stop dynamics if value <=0 for deceleration is configured
                IF (config.fastStop.deceleration <= 0.0) // Read TO emergencyStop deceleration only if fastStop.deceleration <= 0
                THEN
                    // Invalid fastStop dynamics configured - read emergency stop dynamics from TO
                    IF (_refSpeedAxis <> NULL) THEN // Axis type is TO_SpeedAxis or TO_PositioningAxis or TO_SynchronousAxis
                        _instHalt.Deceleration := _refSpeedAxis^.DynamicDefaults.EmergencyDeceleration;
                    ELSE // Invalid TO specification
                        _instHalt.Deceleration := -1.0;
                    END_IF;
                ELSE
                    // Valid fastStop dynamics configured
                    _instHalt.Deceleration := config.fastStop.deceleration;
                END_IF;
                _instHalt.AbortAcceleration := config.fastStop.abortAcceleration; // Use always config
                _instHalt.Jerk := config.fastStop.jerk; // Use always config for jerk value
            END_IF;

            // Call of MC_Command
            _instHalt(Axis := _refSpeedAxis^,
                      Execute := (_basicCommand.%X0 OR _firstCycleBasicMotion));

            // Evaluate MC_Command
            IF (_instHalt.Busy = FALSE) AND
                (_instHalt.Error = FALSE) AND
                (_instHalt.Done = FALSE) AND
                (_instHalt.CommandAborted = FALSE)
            THEN
                // Return to NO_SELECTION if command finished
                _state := AXIS_MOTION;
                _basicMotionState := NO_SELECTION;
                _stopWithoutSignalization := FALSE;

            ELSIF (_instHalt.Done = TRUE) THEN
                IF (_firstCycleDone = TRUE) THEN
                    // Command is reset
                    IF (_instTorqueLimiting.Error = FALSE) // Dont reset error is pending
                    THEN
                        // Reset status not if torquelimiting error is pending
                        IF _stopWithoutSignalization THEN
                            ;
                        ELSE
                            _status := AxisStatus#STATUS_SUBSEQUENT_CALL;
                            _statusText := STRING#'STATUS_SUBSEQUENT_CALL';
                            _errorAutoCleared := FALSE;
                        END_IF;
                    END_IF;

                    _firstCycleDone := FALSE;
                END_IF;

            ELSIF (_instHalt.Error = TRUE) AND (_stopWithoutSignalization = FALSE) // signal the error if fastStop is selected via the input 'fastStop'
            THEN
                // Errorhandling
                _status := AxisStatus#ERR_MC_HALT;
                _statusText := STRING#'ERR_MC_HALT';
                _errorAutoCleared := TRUE;
                _diagnostics.subfunctionStatus := _instHalt.ErrorId;
                _subfunctionStatus := _instHalt.ErrorId;

                IF (config.fastStop.replaceStopPossible = TRUE) THEN
                    // Set next state
                    _basicMotionState := NO_SELECTION;
                END_IF;

            // ELSE
            //   ; // Command selected
            END_IF;

            // Write MC_Command outputs to internal variable
            _exeOfBasicMotion := 0;
            _exeOfBasicMotion.%X0 := _instHalt.Busy;
            _exeOfBasicMotion.%X1 := _instHalt.Done;
            _exeOfBasicMotion.%X2 := _instHalt.CommandAborted;
            _exeOfBasicMotion.%X3 := _instHalt.Error;

        END_IF;

        //----------------------------------------------------------------------------------------------
        // Store values and reset variables
        //----------------------------------------------------------------------------------------------

        // Reset variables to determine first cycle of a new command
        IF (_firstCycleReset = TRUE) THEN
            _firstCycleReset := FALSE;
        END_IF;
        IF (_firstCycleHoming = TRUE) THEN
            _firstCycleHoming := FALSE;
        END_IF;
        _homingOld := tempHoming;

        _firstCycleBasicMotion := FALSE;
        _basicCommandOld := _basicCommand;

        IF (_firstCycleSupImpMotion = TRUE) THEN
            _firstCycleSupImpMotion := FALSE;
        END_IF;
        _supImpCommandOld := _supImpCommand;

        // Store last values for edge detection
        _enableOld := tempEnable;
        _enableAxisOld := tempEnableAxis;
        _extendedCommandOld := _extendedCommand;
        _powerErrorOld := _instPower.Error;

        //----------------------------------------------------------------------------------------------
        // Writing outputs
        //----------------------------------------------------------------------------------------------

        // Writing status outputs
        resetActive := (_resetState = CMD_BUSY);

        IF (_errorUserCleared = TRUE) THEN
            ; // Reset variables at ErrorUserCleared
            _basicMotionState := NO_SELECTION;
            _exeOfBasicMotion := NO_SELECTION;
            _supImpMotionState := NO_SELECTION;
            _exeOfSupImpMotionState := NO_SELECTION;
            _exeOfHoming := NO_SELECTION;
        END_IF;

        IF (config.power.externalMC_PowerCall = FALSE) THEN
            // Generate the 'axisEnabled' status via the status of the MC_Power instance
            IF (_instPower.Status = TRUE) THEN
                // Axis enabled
                axisEnabled := TRUE;

            ELSIF (_instPower.Error = TRUE) AND (_instPower.Status = FALSE) THEN
                // Reset status if error occurred
                axisEnabled := FALSE;

            ELSIF (_instPower.Busy = FALSE) THEN
                // Reset if MC_Power is not busy
                axisEnabled := FALSE;
            END_IF;

        ELSE // (config.power.externalMC_PowerCall = TRUE)
            // Generate the 'axisEnabled' status via StatusWord Bit 0
            axisEnabled := tempStatusWord.%X0; // StatusWord Bit 0: Enable status. The technology object has been enabled
        END_IF;

        // Writing Busy, Done and Aborted outputs for basic motion commands
        IF (_basicMotionState > NO_SELECTION) AND (_basicMotionState <> ACTIVE_HOMING_SELECTED) THEN
            commandBusy := _exeOfBasicMotion.%X0;
            commandDone := _exeOfBasicMotion.%X1;
            commandAborted := _exeOfBasicMotion.%X2;
            inVelocity := _exeOfBasicMotion.%X4;
            inSync := _exeOfBasicMotion.%X7;
            startSync := _exeOfBasicMotion.%X6;
            endOfProfile := _exeOfBasicMotion.%X8;
        ELSE
            commandBusy := FALSE;
            commandDone := FALSE;
            commandAborted := FALSE;
            inVelocity := FALSE;
            inSync := FALSE;
            startSync := FALSE;
            endOfProfile := FALSE;
        END_IF;

        // Writing outputs up to LAxisCtrl_SpeedAxis
        IF (_torqueLimitingState = TORQUE_LIMITING_SELECTED) THEN
            torqueLimitingSelected := TRUE;
        ELSE
            torqueLimitingSelected := FALSE;
        END_IF;

        inLimitation := _instTorqueLimiting.InLimitation;
        fastStopSelected := _basicMotionState.%X0;
        stopSelected := _basicMotionState.%X1;
        jogSelected := _basicMotionState.%X2 OR _basicMotionState.%X3;
        moveVelocitySelected := _basicMotionState.%X4;
        // Writing outputs up to LAxisCtrl_PosAxis
        inClamping := _instTorqueLimiting.InClamping;
        posRelativeSelected := _basicMotionState.%X5;
        posAbsoluteSelected := _basicMotionState.%X6;
        // Writing outputs up to LAxisCtrl_SyncAxisRelGearing
        gearInRelativeSelected := _basicMotionState.%X7;
        // Writing outputs up to LAxisCtrl_SyncAxisCamming
        gearInAbsoluteSelected := _basicMotionState.%X8;
        gearInVelocitySelected := _basicMotionState.%X12;
        camInSelected := _basicMotionState.%X9;
        gearOutCamOutSelected := _basicMotionState.%X11;
        inSimulation := _instSyncMotionSimulation.InSimulation;

        // Writing Busy, Done and Aborted outputs for homing
        IF (_passiveHomingState = STANDARD_HOMING) THEN
            homingSelected := TRUE;
            homingCommandBusy := _exeOfHoming.%X0;
            homingCommandDone := _exeOfHoming.%X1;
            homingCommandAborted := _exeOfHoming.%X2;
        ELSE
            IF (_basicMotionState = ACTIVE_HOMING_SELECTED) THEN
                homingSelected := TRUE;
                homingCommandBusy := _exeOfBasicMotion.%X0;
                homingCommandDone := _exeOfBasicMotion.%X1;
                homingCommandAborted := _exeOfBasicMotion.%X2;
            ELSE
                homingSelected := FALSE;
                homingCommandBusy := FALSE;
                homingCommandDone := FALSE;
                homingCommandAborted := FALSE;
            END_IF;
        END_IF;

        // Writing outputs for superimposed motion commands
        IF (_supImpMotionState <> NO_SELECTION) THEN
            superimposedBusy := _exeOfSupImpMotionState.%X0;
            superimposedDone := _exeOfSupImpMotionState.%X1;
            superimposedAborted := _exeOfSupImpMotionState.%X2;
            superimposedStart := _exeOfSupImpMotionState.%X4;
        ELSE
            superimposedBusy := FALSE;
            superimposedDone := FALSE;
            superimposedAborted := FALSE;
            superimposedStart := FALSE;
        END_IF;

        posSuperimposedSelected := _supImpMotionState.%X0;
        haltSuperimposedSelected := _supImpMotionState.%X3;
        phasingSelected := _supImpMotionState.%X1;
        offsetSelected := _supImpMotionState.%X2;

        //----------------------------------------------------------------------------------------------
        // Error handling
        //----------------------------------------------------------------------------------------------

        IF _errorUserCleared THEN
            valid := FALSE;
            busy := TRUE;
            error := TRUE;
            subfunctionStatus := _subfunctionStatus;
            _diagnostics.status := _status;

        ELSIF _errorAutoCleared THEN
            valid := FALSE;
            busy := TRUE;
            error := TRUE;
            subfunctionStatus := _subfunctionStatus;
            _diagnostics.status := _status;

        ELSE
            // Process normal output values
            valid := TRUE;
            error := FALSE;
            subfunctionStatus := WORD#16#0000;
            _subfunctionStatus := WORD#16#0000;
        END_IF;

        status := _status;

        IF (_status <> _statusOld) THEN
            statusText := _statusText;
            diagnostics := _diagnostics;
        END_IF;

        // Edge detection
        _statusOld := _status;

    END_FUNCTION_BLOCK
END_NAMESPACE
